// TIA Portal V16 export
// export: Created 2023-03-29T11:03:27.4951312Z, ExportSetting WithDefaults, DisplayName Totally Integrated Automation Portal, DisplayVersion V16 Update 6, DisplayName TIA Portal Version Control Interface, DisplayVersion V16 Update 2, DisplayName TIA Portal Openness, DisplayVersion V16 Update 6, DisplayName STEP 7 Professional, DisplayVersion V16 Update 6, DisplayName STEP 7 Safety, DisplayVersion V16, DisplayName WinCC Advanced, DisplayVersion V16 Update 6
FUNCTION "Saving_Canged_Data_Word_USInt" : Void   // FC38, LAD
{ S7_Optimized_Access := 'TRUE' }
AUTHOR : rtecmer
VERSION : 0.1
// Funkcj po sprawdzeniu czy dane w pobranym bloku różnią się od danyc w bloku SCADA dokonuje operacji zapisu jeśli byatąpiła różnica danych.
// stored: AutoNumber false, IsIECCheckEnabled false, SetENOAutomatically false, UDAEnableTagReadback false
   VAR_IN_OUT
      "dbHold_download.sterowanie" : USInt;   // Zmienna zadawana i porównywana
      "DB10_instance_SCADA." : USInt;   // Zmienna do porównania
      memTrig_Client_Receiving_ : Bool;   // pamięć zbocze zmiany
   END_VAR
   VAR_TEMP
      dbHold_download : Int;
   END_VAR
   VAR_TEMP   // added for the SCL form of the ladder/FBD networks
      _w1 : Bool;
      _w2 : Bool;
   END_VAR
BEGIN

REGION Network 2
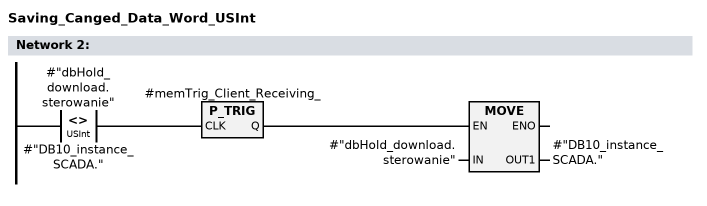
   RUNG wire#powerrail
      { S7_Templates := "SrcType := USInt" } NE_Contact(in1 := #"dbHold_download.sterowanie", in2 := #"DB10_instance_SCADA.")
      P_Trig( #memTrig_Client_Receiving_ )
      Move(in := #"dbHold_download.sterowanie", out1 => #"DB10_instance_SCADA.")
   END_RUNG
   // the same network as SCL:
   #_w1 := #"dbHold_download.sterowanie" <> #"DB10_instance_SCADA.";
   #_w2 := #_w1 AND NOT #memTrig_Client_Receiving_;   // rising edge
   #memTrig_Client_Receiving_ := #_w1;
   IF #_w2 THEN #"DB10_instance_SCADA." := #"dbHold_download.sterowanie"; END_IF;
END_REGION
END_FUNCTION
